SUBAPPLICATION IX_TO_Aux_QX (* logiBUS_IX auf isobus Aux_QX (generisch), event-basiert *)
  (* Standard: 61499-2 *)
  (* Version 1.0, 2026-09-09, Franz Höpfinger, Meisterschulen am Ostbahnhof, Ausgelagert aus Uebung_003c_sub zur Wiederverwendung. *)
  PACKAGE MyLib::sys;
  IMPORT logiBUS::io::DI::logiBUS_DI::Invalid;
  IMPORT logiBUS::io::DI::logiBUS_DI_S;
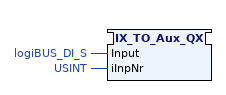
  VAR_INPUT
    Input : logiBUS::io::DI::logiBUS_DI_S := Invalid; (* Identify the Input Input_I1..I8 *)
    iInpNr : USINT := 0; (* Number of auxiliary array - corresponds with the order in the pool that means first aux input in pool is iInpNr = 0 etc. *)
  END_VAR
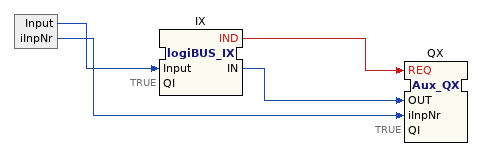
  FBS
    QX : isobus::UT::io::Auxiliary::OUT::Aux_QX(QI := TRUE);
    IX : logiBUS::io::DI::logiBUS_IX(QI := TRUE);
  END_FBS
  EVENT_CONNECTIONS
    IX.IND TO QX.REQ;
  END_CONNECTIONS
  DATA_CONNECTIONS
    IX.IN TO QX.OUT;
    Input TO IX.Input;
    iInpNr TO QX.iInpNr;
  END_CONNECTIONS
END_SUBAPPLICATION
